PROGRAM ClearScript
VAR
END_VAR

IF GVL_MOTION.EXT_CTR.CMDCLR THEN
	GVL_MOTION.EXT_CTR.CMDCLR	:= FALSE;
	GVL_MOTION.EXT_CTR.CMDRUN 	:= FALSE;
	GVL_MOTION.ScriptEnd 		:= 0;
	GVL_MOTION.CurInstruction 	:= 0;
	GVL_MOTION.InstructionState := 0;
	GVL_MOTION.HaltMem 			:= FALSE;
	GVL_MOTION.TxtBxWaitOK 		:= TRUE;
	MEMSET(ADR(GVL_MOTION.Script), 0, SIZEOF(GVL_MOTION.Script));
END_IF

END_PROGRAM

(* stored: Version 1.1.0.1, ProductVersion 3.1.4026.18
   POU ClearScript: Id {ea9c4e96-dc01-4bcf-937a-581bfdc2a510}, SpecialFunc None *)
